VAR_GLOBAL
	gbKin : KinematicsD4;
END_VAR

(* stored: Version 1.1.0.1, ProductVersion 3.1.4024.11
   GVL GVL_Kinematics: Id {89b5f3d8-491e-4db3-8966-ac19de6bd777} *)
